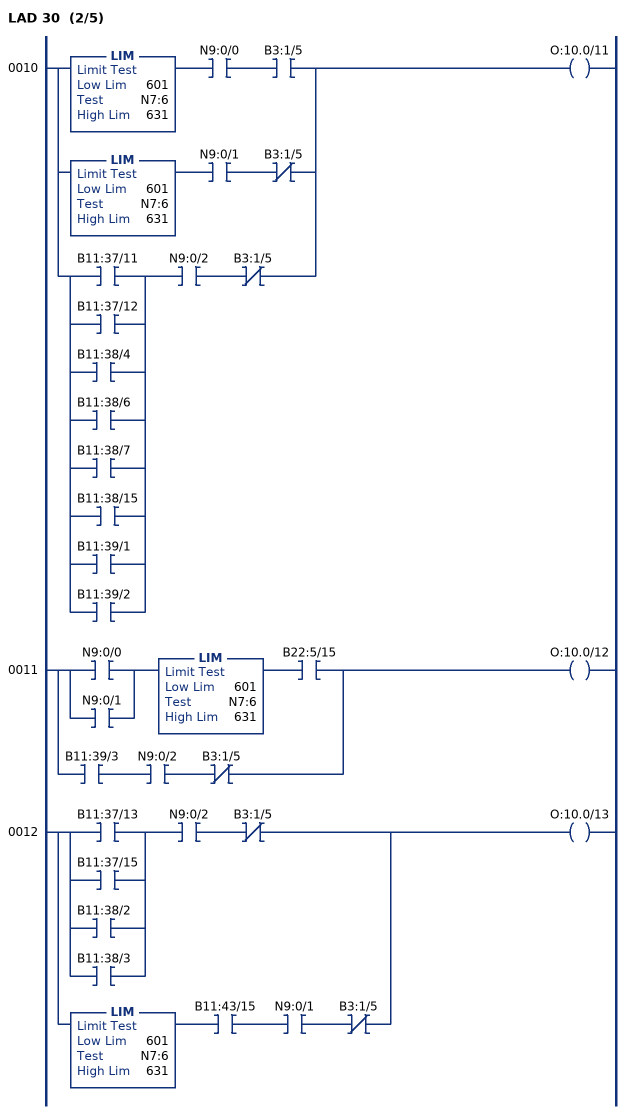
% Rung: 10 %
SOR BST LIM 601 N7:6 631 XIC N9:0/0 XIC B3:1/5 NXB LIM 601 N7:6 631 XIC N9:0/1 XIO B3:1/5 NXB BST XIC B11:37/11 NXB XIC B11:37/12 NXB XIC B11:38/4 NXB XIC B11:38/6 NXB XIC B11:38/7 NXB XIC B11:38/15 NXB XIC B11:39/1 NXB XIC B11:39/2 BND XIC N9:0/2 XIO B3:1/5 BND OTE O:10.0/11 EOR
% Rung: 11 %
SOR BST BST XIC N9:0/0 NXB XIC N9:0/1 BND LIM 601 N7:6 631 XIC B22:5/15 NXB XIC B11:39/3 XIC N9:0/2 XIO B3:1/5 BND OTE O:10.0/12 EOR
% Rung: 12 %
SOR BST BST XIC B11:37/13 NXB XIC B11:37/15 NXB XIC B11:38/2 NXB XIC B11:38/3 BND XIC N9:0/2 XIO B3:1/5 NXB LIM 601 N7:6 631 XIC B11:43/15 XIC N9:0/1 XIO B3:1/5 BND OTE O:10.0/13 EOR

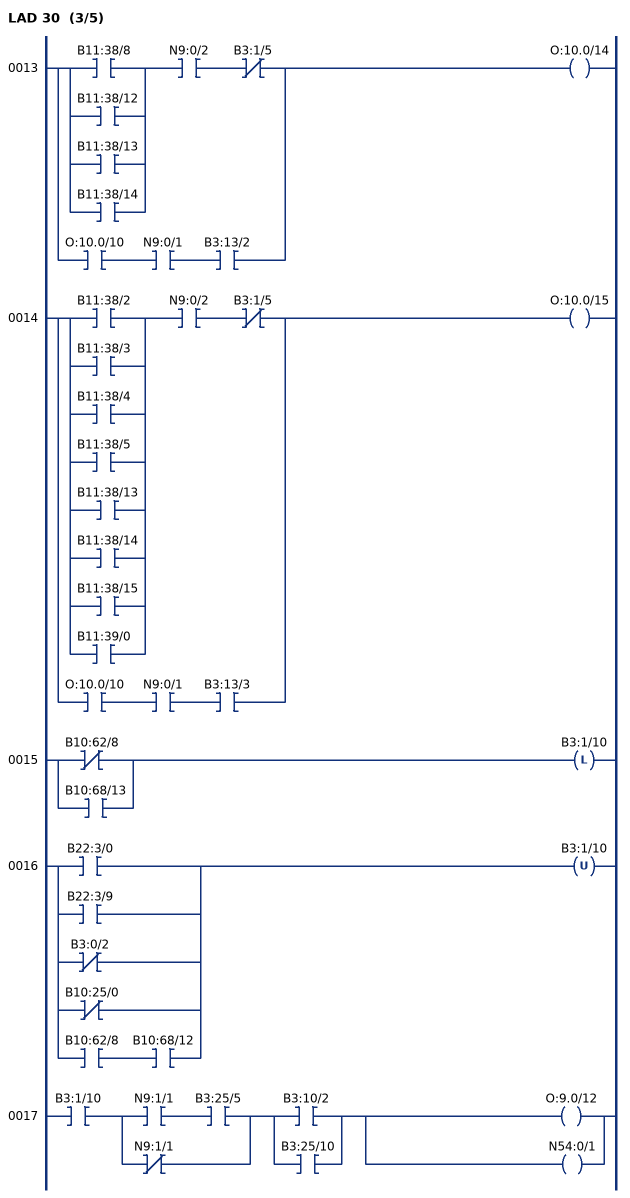
% Rung: 13 %
SOR BST BST XIC B11:38/8 NXB XIC B11:38/12 NXB XIC B11:38/13 NXB XIC B11:38/14 BND XIC N9:0/2 XIO B3:1/5 NXB XIC O:10.0/10 XIC N9:0/1 XIC B3:13/2 BND OTE O:10.0/14 EOR
% Rung: 14 %
SOR BST BST XIC B11:38/2 NXB XIC B11:38/3 NXB XIC B11:38/4 NXB XIC B11:38/5 NXB XIC B11:38/13 NXB XIC B11:38/14 NXB XIC B11:38/15 NXB XIC B11:39/0 BND XIC N9:0/2 XIO B3:1/5 NXB XIC O:10.0/10 XIC N9:0/1 XIC B3:13/3 BND OTE O:10.0/15 EOR
% Rung: 15 %
SOR BST XIO B10:62/8 NXB XIC B10:68/13 BND OTL B3:1/10 EOR
% Rung: 16 %
SOR BST XIC B22:3/0 NXB XIC B22:3/9 NXB XIO B3:0/2 NXB XIO B10:25/0 NXB XIC B10:62/8 XIC B10:68/12 BND OTU B3:1/10 EOR
% Rung: 17 %
SOR XIC B3:1/10 BST XIC N9:1/1 XIC B3:25/5 NXB XIO N9:1/1 BND BST XIC B3:10/2 NXB XIC B3:25/10 BND BST OTE O:9.0/12 NXB OTE N54:0/1 BND EOR

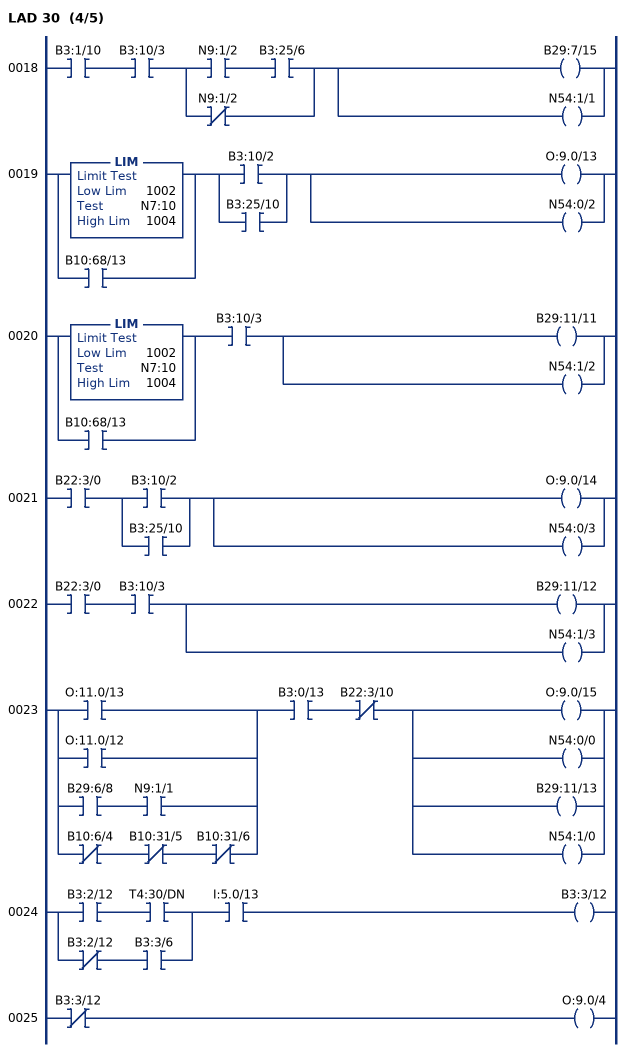
% Rung: 18 %
SOR XIC B3:1/10 XIC B3:10/3 BST XIC N9:1/2 XIC B3:25/6 NXB XIO N9:1/2 BND BST OTE B29:7/15 NXB OTE N54:1/1 BND EOR
% Rung: 19 %
SOR BST LIM 1002 N7:10 1004 NXB XIC B10:68/13 BND BST XIC B3:10/2 NXB XIC B3:25/10 BND BST OTE O:9.0/13 NXB OTE N54:0/2 BND EOR
% Rung: 20 %
SOR BST LIM 1002 N7:10 1004 NXB XIC B10:68/13 BND XIC B3:10/3 BST OTE B29:11/11 NXB OTE N54:1/2 BND EOR
% Rung: 21 %
SOR XIC B22:3/0 BST XIC B3:10/2 NXB XIC B3:25/10 BND BST OTE O:9.0/14 NXB OTE N54:0/3 BND EOR
% Rung: 22 %
SOR XIC B22:3/0 XIC B3:10/3 BST OTE B29:11/12 NXB OTE N54:1/3 BND EOR
% Rung: 23 %
SOR BST BST XIC O:11.0/13 NXB XIC O:11.0/12 BND NXB XIC B29:6/8 XIC N9:1/1 NXB XIO B10:6/4 XIO B10:31/5 XIO B10:31/6 BND XIC B3:0/13 XIO B22:3/10 BST OTE O:9.0/15 NXB OTE N54:0/0 NXB OTE B29:11/13 NXB OTE N54:1/0 BND EOR
% Rung: 24 %
SOR BST XIC B3:2/12 XIC T4:30/DN NXB XIO B3:2/12 XIC B3:3/6 BND XIC I:5.0/13 OTE B3:3/12 EOR
% Rung: 25 %
SOR XIO B3:3/12 OTE O:9.0/4 EOR

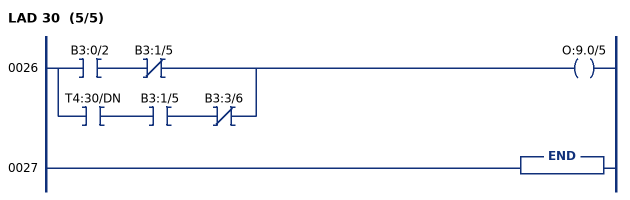
% Rung: 26 %
SOR BST XIC B3:0/2 XIO B3:1/5 NXB XIC T4:30/DN XIC B3:1/5 XIO B3:3/6 BND OTE O:9.0/5 EOR
% Rung: 27 %
SOR END EOR

LADDER 31
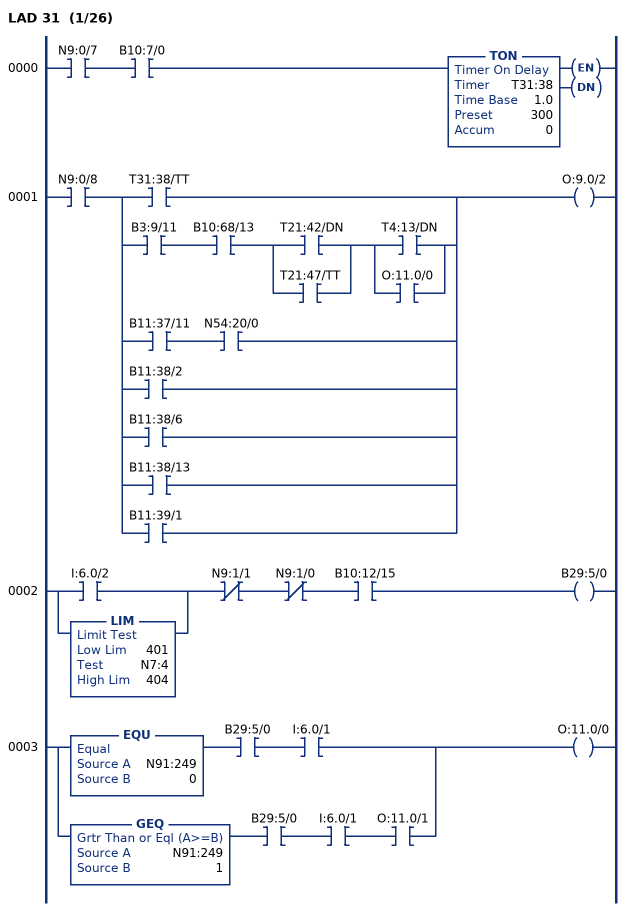
% Rung: 0 %
SOR XIC N9:0/7 XIC B10:7/0 TON T31:38 1.0 300 0 EOR
% Rung: 1 %
SOR XIC N9:0/8 BST XIC T31:38/TT NXB XIC B3:9/11 XIC B10:68/13 BST XIC T21:42/DN NXB XIC T21:47/TT BND BST XIC T4:13/DN NXB XIC O:11.0/0 BND NXB XIC B11:37/11 XIC N54:20/0 NXB XIC B11:38/2 NXB XIC B11:38/6 NXB XIC B11:38/13 NXB XIC B11:39/1 BND OTE O:9.0/2 EOR
% Rung: 2 %
SOR BST XIC I:6.0/2 NXB LIM 401 N7:4 404 BND XIO N9:1/1 XIO N9:1/0 XIC B10:12/15 OTE B29:5/0 EOR
% Rung: 3 %
SOR BST EQU N91:249 0 XIC B29:5/0 XIC I:6.0/1 NXB GEQ N91:249 1 XIC B29:5/0 XIC I:6.0/1 XIC O:11.0/1 BND OTE O:11.0/0 EOR

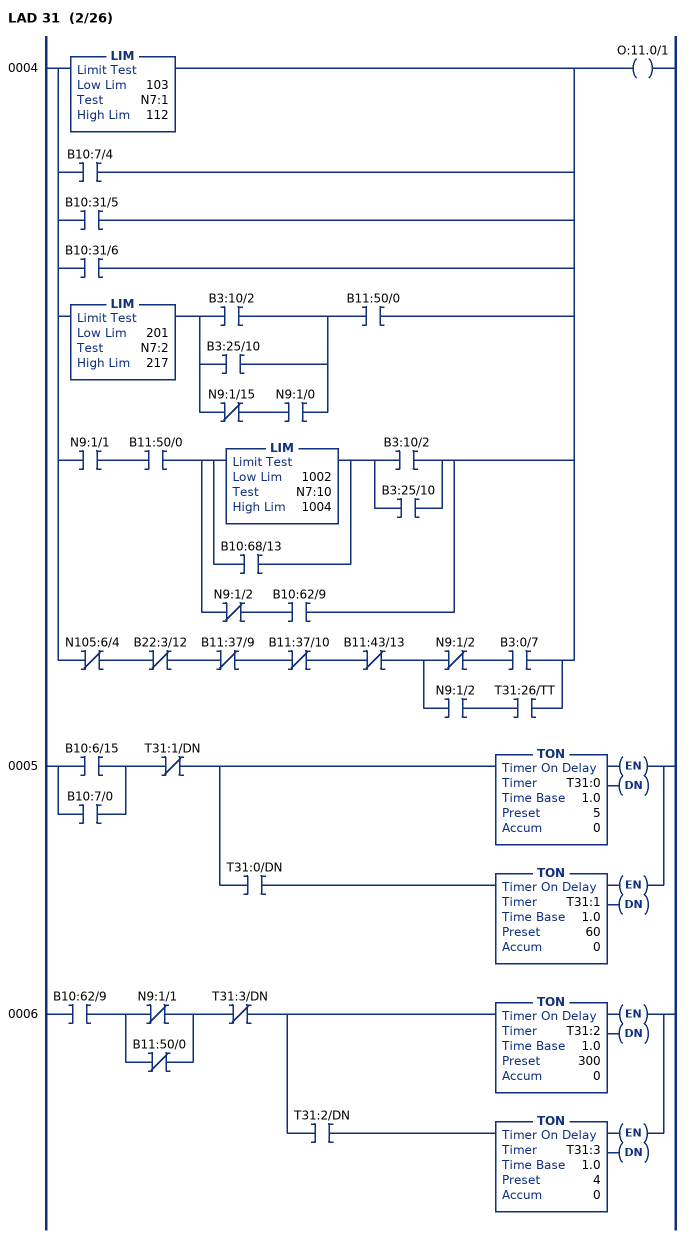
% Rung: 4 %
SOR BST LIM 103 N7:1 112 NXB XIC B10:7/4 NXB XIC B10:31/5 NXB XIC B10:31/6 NXB LIM 201 N7:2 217 BST XIC B3:10/2 NXB XIC B3:25/10 NXB XIO N9:1/15 XIC N9:1/0 BND XIC B11:50/0 NXB XIC N9:1/1 XIC B11:50/0 BST BST LIM 1002 N7:10 1004 NXB XIC B10:68/13 BND BST XIC B3:10/2 NXB XIC B3:25/10 BND NXB XIO N9:1/2 XIC B10:62/9 BND NXB XIO N105:6/4 XIO B22:3/12 XIO B11:37/9 XIO B11:37/10 XIO B11:43/13 BST XIO N9:1/2 XIC B3:0/7 NXB XIC N9:1/2 XIC T31:26/TT BND BND OTE O:11.0/1 EOR
% Rung: 5 %
SOR BST XIC B10:6/15 NXB XIC B10:7/0 BND XIO T31:1/DN BST TON T31:0 1.0 5 0 NXB XIC T31:0/DN TON T31:1 1.0 60 0 BND EOR
% Rung: 6 %
SOR XIC B10:62/9 BST XIO N9:1/1 NXB XIO B11:50/0 BND XIO T31:3/DN BST TON T31:2 1.0 300 0 NXB XIC T31:2/DN TON T31:3 1.0 4 0 BND EOR

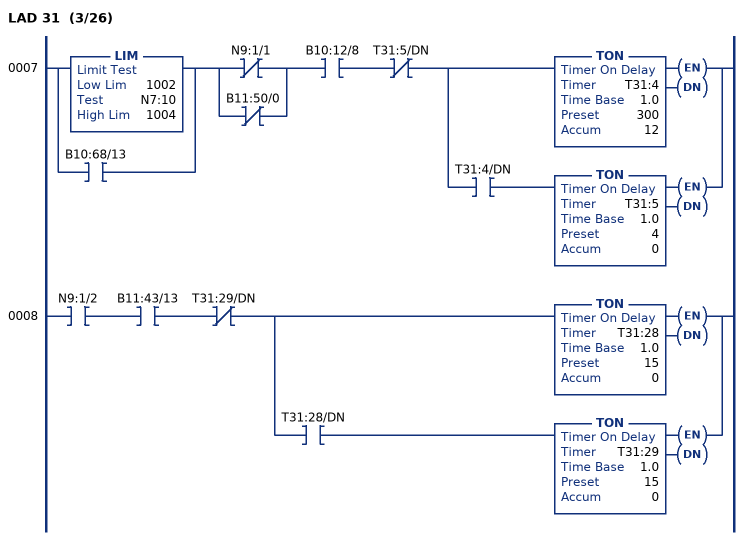
% Rung: 7 %
SOR BST LIM 1002 N7:10 1004 NXB XIC B10:68/13 BND BST XIO N9:1/1 NXB XIO B11:50/0 BND XIC B10:12/8 XIO T31:5/DN BST TON T31:4 1.0 300 12 NXB XIC T31:4/DN TON T31:5 1.0 4 0 BND EOR
% Rung: 8 %
SOR XIC N9:1/2 XIC B11:43/13 XIO T31:29/DN BST TON T31:28 1.0 15 0 NXB XIC T31:28/DN TON T31:29 1.0 15 0 BND EOR

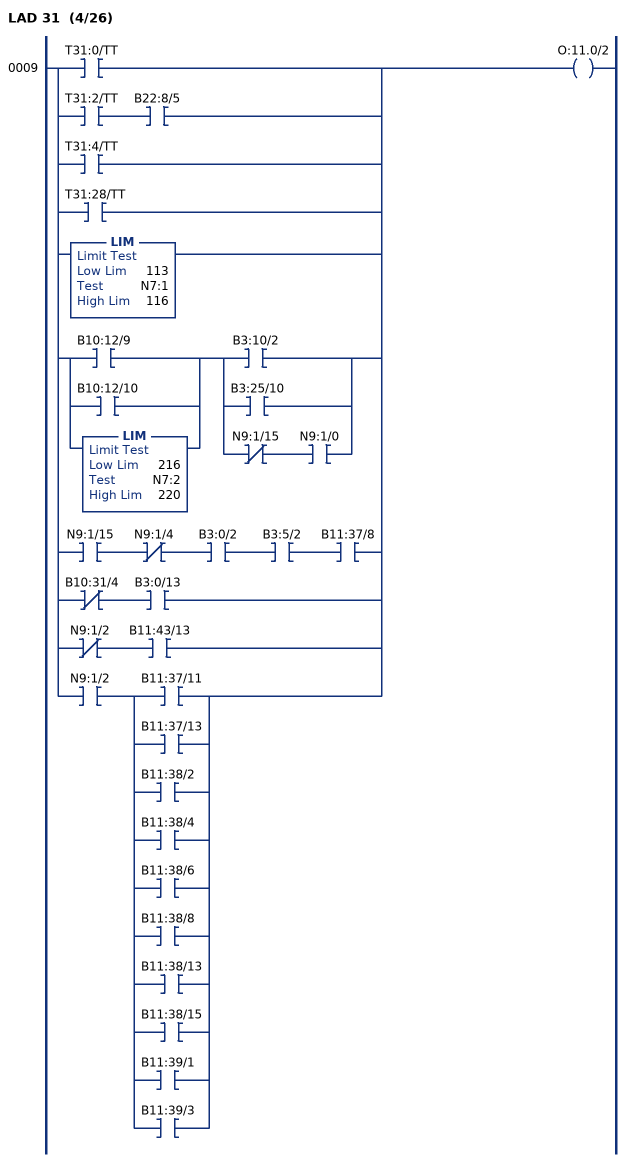
% Rung: 9 %
SOR BST XIC T31:0/TT NXB XIC T31:2/TT XIC B22:8/5 NXB XIC T31:4/TT NXB XIC T31:28/TT NXB LIM 113 N7:1 116 NXB BST XIC B10:12/9 NXB XIC B10:12/10 NXB LIM 216 N7:2 220 BND BST XIC B3:10/2 NXB XIC B3:25/10 NXB XIO N9:1/15 XIC N9:1/0 BND NXB XIC N9:1/15 XIO N9:1/4 XIC B3:0/2 XIC B3:5/2 XIC B11:37/8 NXB XIO B10:31/4 XIC B3:0/13 NXB XIO N9:1/2 XIC B11:43/13 NXB XIC N9:1/2 BST XIC B11:37/11 NXB XIC B11:37/13 NXB XIC B11:38/2 NXB XIC B11:38/4 NXB XIC B11:38/6 NXB XIC B11:38/8 NXB XIC B11:38/13 NXB XIC B11:38/15 NXB XIC B11:39/1 NXB XIC B11:39/3 BND BND OTE O:11.0/2 EOR

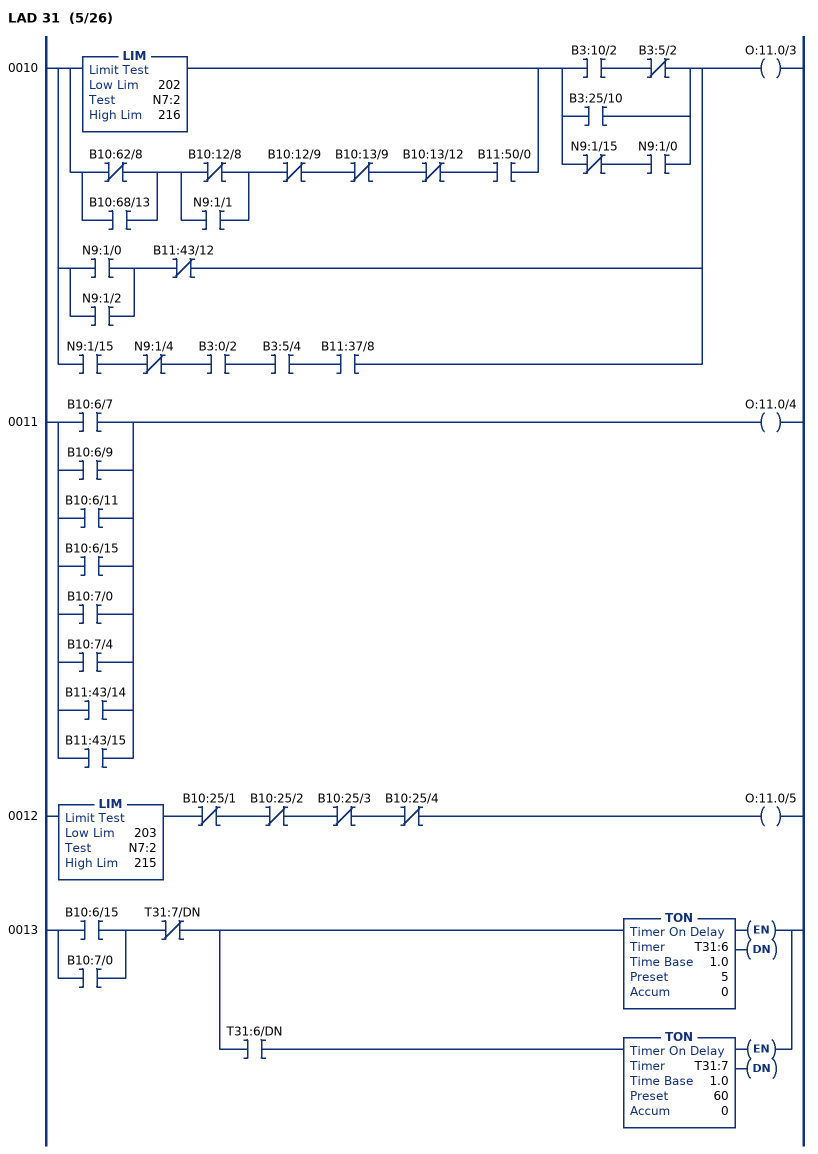
% Rung: 10 %
SOR BST BST LIM 202 N7:2 216 NXB BST XIO B10:62/8 NXB XIC B10:68/13 BND BST XIO B10:12/8 NXB XIC N9:1/1 BND XIO B10:12/9 XIO B10:13/9 XIO B10:13/12 XIC B11:50/0 BND BST XIC B3:10/2 XIO B3:5/2 NXB XIC B3:25/10 NXB XIO N9:1/15 XIC N9:1/0 BND NXB BST XIC N9:1/0 NXB XIC N9:1/2 BND XIO B11:43/12 NXB XIC N9:1/15 XIO N9:1/4 XIC B3:0/2 XIC B3:5/4 XIC B11:37/8 BND OTE O:11.0/3 EOR
% Rung: 11 %
SOR BST XIC B10:6/7 NXB XIC B10:6/9 NXB XIC B10:6/11 NXB XIC B10:6/15 NXB XIC B10:7/0 NXB XIC B10:7/4 NXB XIC B11:43/14 NXB XIC B11:43/15 BND OTE O:11.0/4 EOR
% Rung: 12 %
SOR LIM 203 N7:2 215 XIO B10:25/1 XIO B10:25/2 XIO B10:25/3 XIO B10:25/4 OTE O:11.0/5 EOR
% Rung: 13 %
SOR BST XIC B10:6/15 NXB XIC B10:7/0 BND XIO T31:7/DN BST TON T31:6 1.0 5 0 NXB XIC T31:6/DN TON T31:7 1.0 60 0 BND EOR

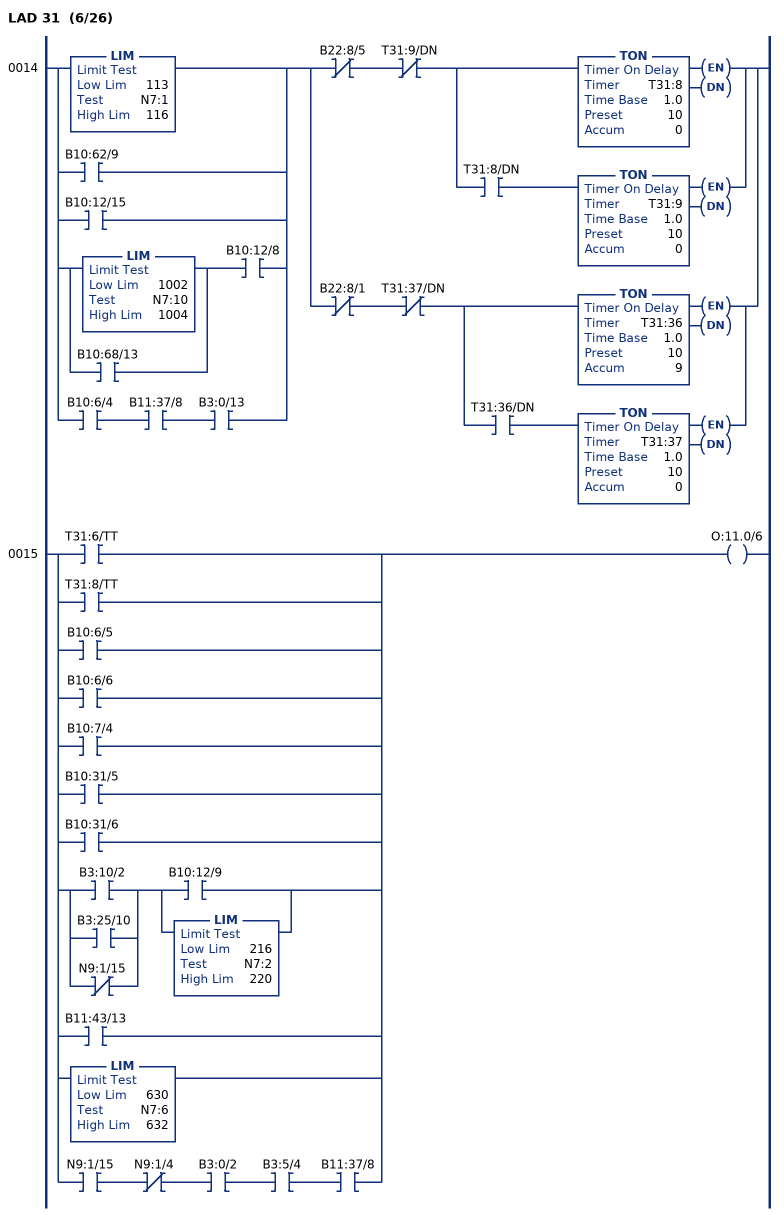
% Rung: 14 %
SOR BST LIM 113 N7:1 116 NXB XIC B10:62/9 NXB XIC B10:12/15 NXB BST LIM 1002 N7:10 1004 NXB XIC B10:68/13 BND XIC B10:12/8 NXB XIC B10:6/4 XIC B11:37/8 XIC B3:0/13 BND BST XIO B22:8/5 XIO T31:9/DN BST TON T31:8 1.0 10 0 NXB XIC T31:8/DN TON T31:9 1.0 10 0 BND NXB XIO B22:8/1 XIO T31:37/DN BST TON T31:36 1.0 10 9 NXB XIC T31:36/DN TON T31:37 1.0 10 0 BND BND EOR
% Rung: 15 %
SOR BST XIC T31:6/TT NXB XIC T31:8/TT NXB XIC B10:6/5 NXB XIC B10:6/6 NXB XIC B10:7/4 NXB XIC B10:31/5 NXB XIC B10:31/6 NXB BST XIC B3:10/2 NXB XIC B3:25/10 NXB XIO N9:1/15 BND BST XIC B10:12/9 NXB LIM 216 N7:2 220 BND NXB XIC B11:43/13 NXB LIM 630 N7:6 632 NXB XIC N9:1/15 XIO N9:1/4 XIC B3:0/2 XIC B3:5/4 XIC B11:37/8 BND OTE O:11.0/6 EOR

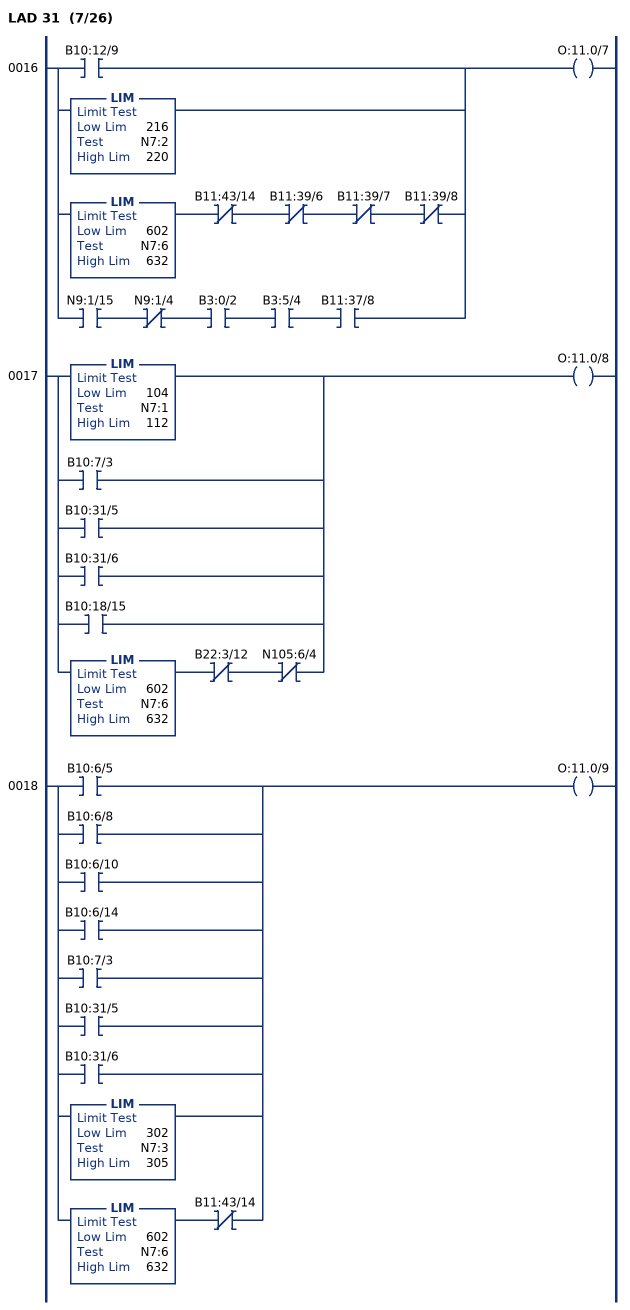
% Rung: 16 %
SOR BST XIC B10:12/9 NXB LIM 216 N7:2 220 NXB LIM 602 N7:6 632 XIO B11:43/14 XIO B11:39/6 XIO B11:39/7 XIO B11:39/8 NXB XIC N9:1/15 XIO N9:1/4 XIC B3:0/2 XIC B3:5/4 XIC B11:37/8 BND OTE O:11.0/7 EOR
% Rung: 17 %
SOR BST LIM 104 N7:1 112 NXB XIC B10:7/3 NXB XIC B10:31/5 NXB XIC B10:31/6 NXB XIC B10:18/15 NXB LIM 602 N7:6 632 XIO B22:3/12 XIO N105:6/4 BND OTE O:11.0/8 EOR
% Rung: 18 %
SOR BST XIC B10:6/5 NXB XIC B10:6/8 NXB XIC B10:6/10 NXB XIC B10:6/14 NXB XIC B10:7/3 NXB XIC B10:31/5 NXB XIC B10:31/6 NXB LIM 302 N7:3 305 NXB LIM 602 N7:6 632 XIO B11:43/14 BND OTE O:11.0/9 EOR

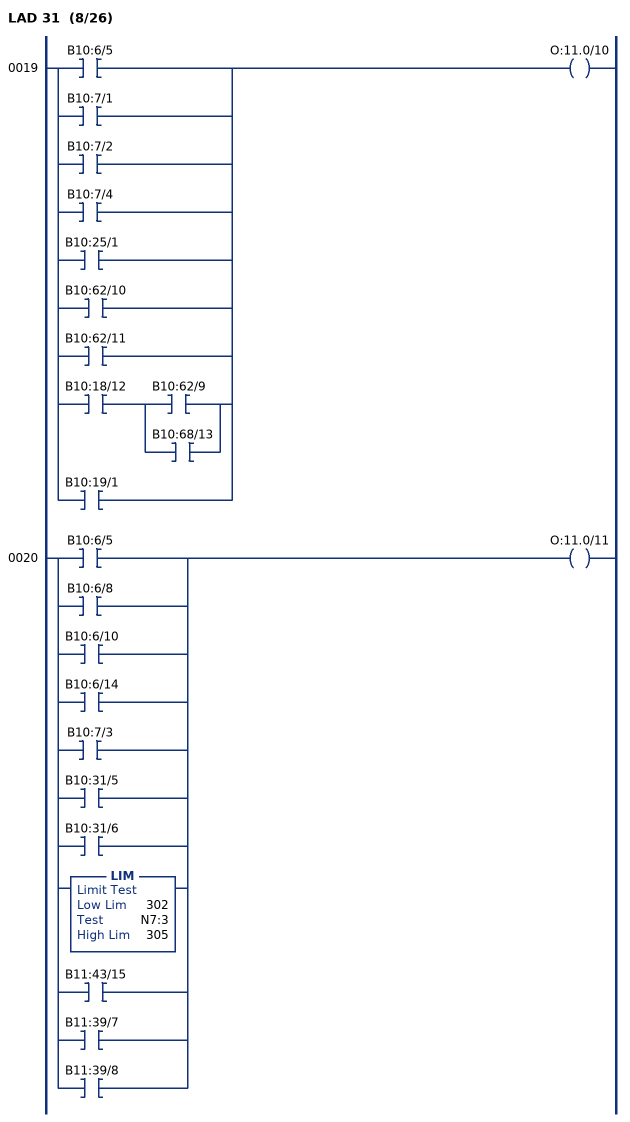
% Rung: 19 %
SOR BST XIC B10:6/5 NXB XIC B10:7/1 NXB XIC B10:7/2 NXB XIC B10:7/4 NXB XIC B10:25/1 NXB XIC B10:62/10 NXB XIC B10:62/11 NXB XIC B10:18/12 BST XIC B10:62/9 NXB XIC B10:68/13 BND NXB XIC B10:19/1 BND OTE O:11.0/10 EOR
% Rung: 20 %
SOR BST XIC B10:6/5 NXB XIC B10:6/8 NXB XIC B10:6/10 NXB XIC B10:6/14 NXB XIC B10:7/3 NXB XIC B10:31/5 NXB XIC B10:31/6 NXB LIM 302 N7:3 305 NXB XIC B11:43/15 NXB XIC B11:39/7 NXB XIC B11:39/8 BND OTE O:11.0/11 EOR

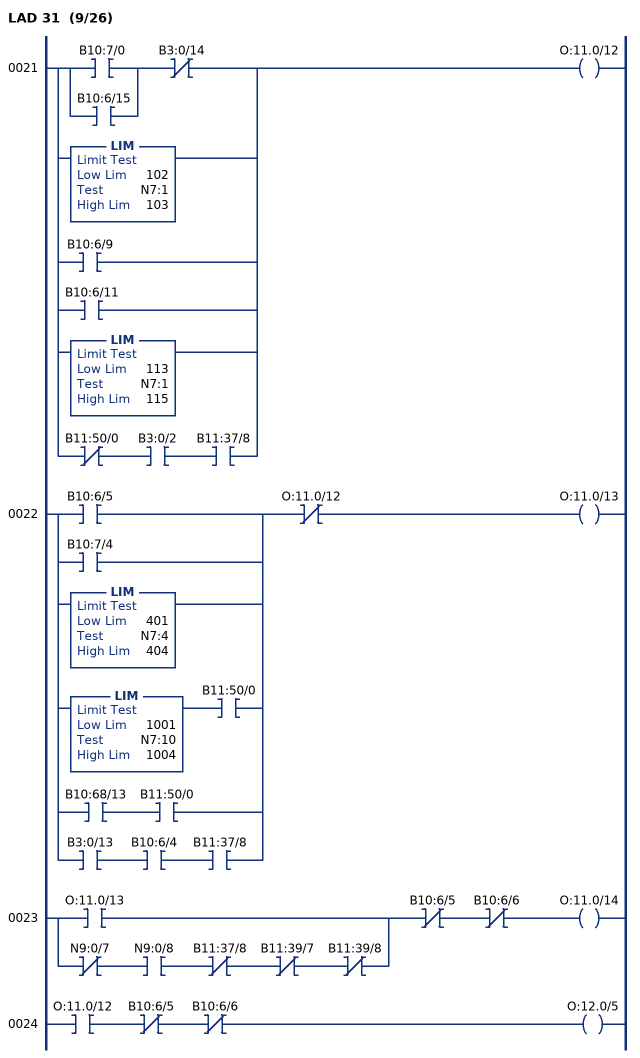
% Rung: 21 %
SOR BST BST XIC B10:7/0 NXB XIC B10:6/15 BND XIO B3:0/14 NXB LIM 102 N7:1 103 NXB XIC B10:6/9 NXB XIC B10:6/11 NXB LIM 113 N7:1 115 NXB XIO B11:50/0 XIC B3:0/2 XIC B11:37/8 BND OTE O:11.0/12 EOR
% Rung: 22 %
SOR BST XIC B10:6/5 NXB XIC B10:7/4 NXB LIM 401 N7:4 404 NXB LIM 1001 N7:10 1004 XIC B11:50/0 NXB XIC B10:68/13 XIC B11:50/0 NXB XIC B3:0/13 XIC B10:6/4 XIC B11:37/8 BND XIO O:11.0/12 OTE O:11.0/13 EOR
% Rung: 23 %
SOR BST XIC O:11.0/13 NXB XIO N9:0/7 XIC N9:0/8 XIO B11:37/8 XIO B11:39/7 XIO B11:39/8 BND XIO B10:6/5 XIO B10:6/6 OTE O:11.0/14 EOR
% Rung: 24 %
SOR XIC O:11.0/12 XIO B10:6/5 XIO B10:6/6 OTE O:12.0/5 EOR

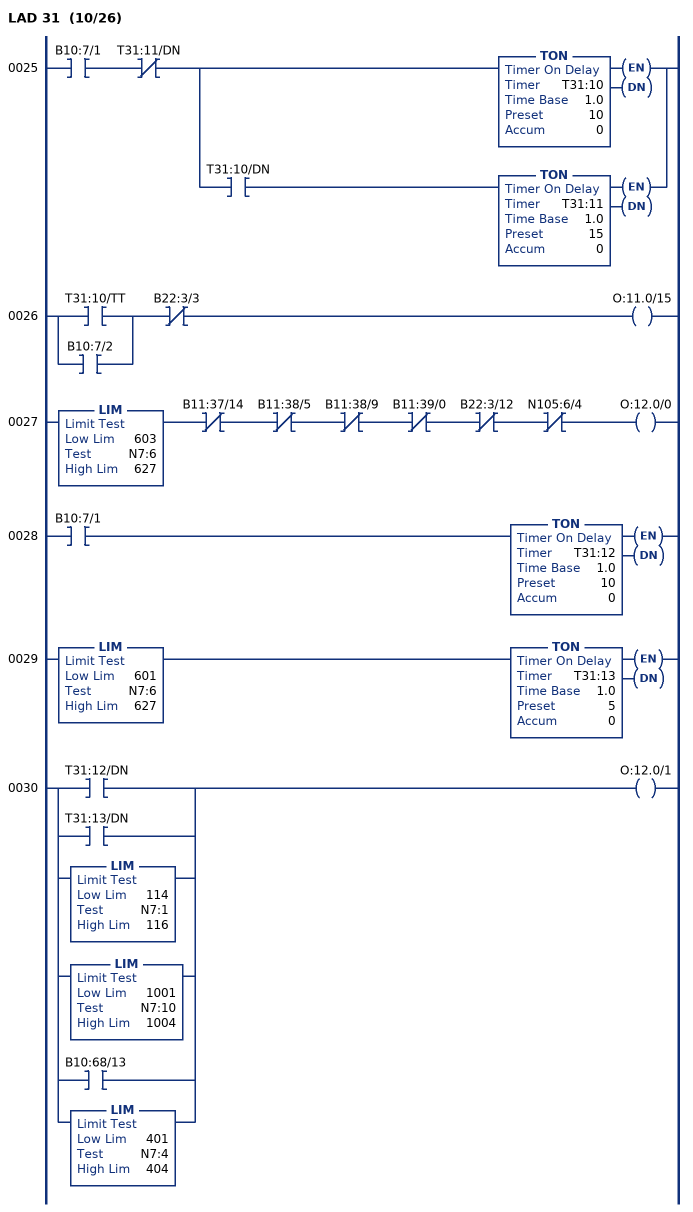
% Rung: 25 %
SOR XIC B10:7/1 XIO T31:11/DN BST TON T31:10 1.0 10 0 NXB XIC T31:10/DN TON T31:11 1.0 15 0 BND EOR
% Rung: 26 %
SOR BST XIC T31:10/TT NXB XIC B10:7/2 BND XIO B22:3/3 OTE O:11.0/15 EOR
% Rung: 27 %
SOR LIM 603 N7:6 627 XIO B11:37/14 XIO B11:38/5 XIO B11:38/9 XIO B11:39/0 XIO B22:3/12 XIO N105:6/4 OTE O:12.0/0 EOR
% Rung: 28 %
SOR XIC B10:7/1 TON T31:12 1.0 10 0 EOR
% Rung: 29 %
SOR LIM 601 N7:6 627 TON T31:13 1.0 5 0 EOR
% Rung: 30 %
SOR BST XIC T31:12/DN NXB XIC T31:13/DN NXB LIM 114 N7:1 116 NXB LIM 1001 N7:10 1004 NXB XIC B10:68/13 NXB LIM 401 N7:4 404 BND OTE O:12.0/1 EOR

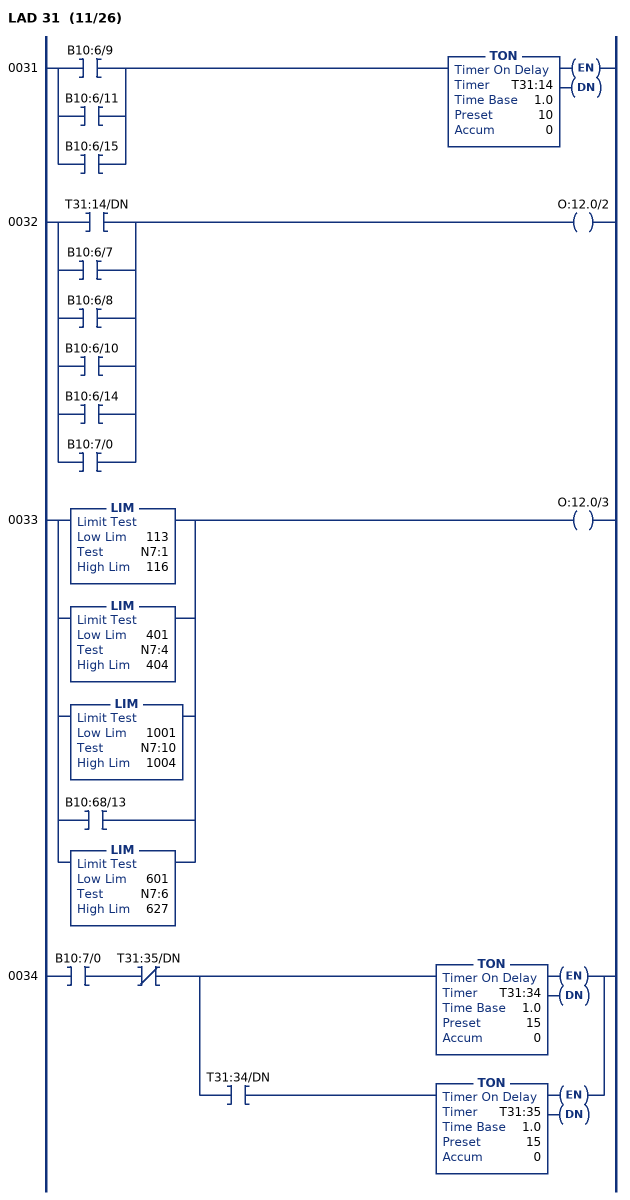
% Rung: 31 %
SOR BST XIC B10:6/9 NXB XIC B10:6/11 NXB XIC B10:6/15 BND TON T31:14 1.0 10 0 EOR
% Rung: 32 %
SOR BST XIC T31:14/DN NXB XIC B10:6/7 NXB XIC B10:6/8 NXB XIC B10:6/10 NXB XIC B10:6/14 NXB XIC B10:7/0 BND OTE O:12.0/2 EOR
% Rung: 33 %
SOR BST LIM 113 N7:1 116 NXB LIM 401 N7:4 404 NXB LIM 1001 N7:10 1004 NXB XIC B10:68/13 NXB LIM 601 N7:6 627 BND OTE O:12.0/3 EOR
% Rung: 34 %
SOR XIC B10:7/0 XIO T31:35/DN BST TON T31:34 1.0 15 0 NXB XIC T31:34/DN TON T31:35 1.0 15 0 BND EOR

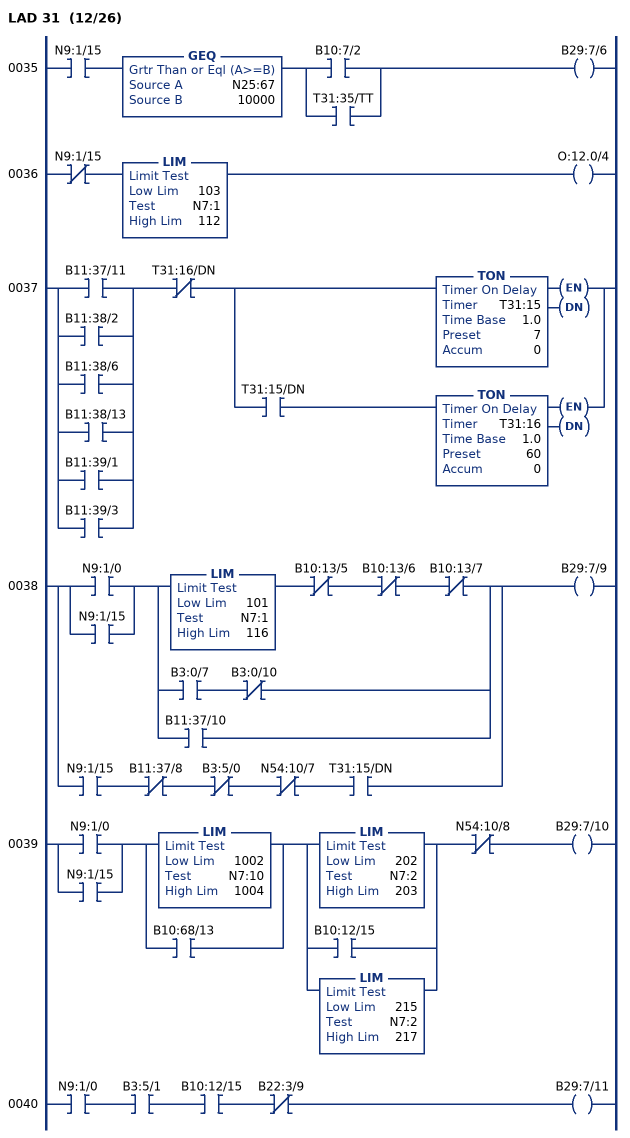
% Rung: 35 %
SOR XIC N9:1/15 GEQ N25:67 10000 BST XIC B10:7/2 NXB XIC T31:35/TT BND OTE B29:7/6 EOR
% Rung: 36 %
SOR XIO N9:1/15 LIM 103 N7:1 112 OTE O:12.0/4 EOR
% Rung: 37 %
SOR BST XIC B11:37/11 NXB XIC B11:38/2 NXB XIC B11:38/6 NXB XIC B11:38/13 NXB XIC B11:39/1 NXB XIC B11:39/3 BND XIO T31:16/DN BST TON T31:15 1.0 7 0 NXB XIC T31:15/DN TON T31:16 1.0 60 0 BND EOR
% Rung: 38 %
SOR BST BST XIC N9:1/0 NXB XIC N9:1/15 BND BST LIM 101 N7:1 116 XIO B10:13/5 XIO B10:13/6 XIO B10:13/7 NXB XIC B3:0/7 XIO B3:0/10 NXB XIC B11:37/10 BND NXB XIC N9:1/15 XIO B11:37/8 XIO B3:5/0 XIO N54:10/7 XIC T31:15/DN BND OTE B29:7/9 EOR
% Rung: 39 %
SOR BST XIC N9:1/0 NXB XIC N9:1/15 BND BST LIM 1002 N7:10 1004 NXB XIC B10:68/13 BND BST LIM 202 N7:2 203 NXB XIC B10:12/15 NXB LIM 215 N7:2 217 BND XIO N54:10/8 OTE B29:7/10 EOR
% Rung: 40 %
SOR XIC N9:1/0 XIC B3:5/1 XIC B10:12/15 XIO B22:3/9 OTE B29:7/11 EOR

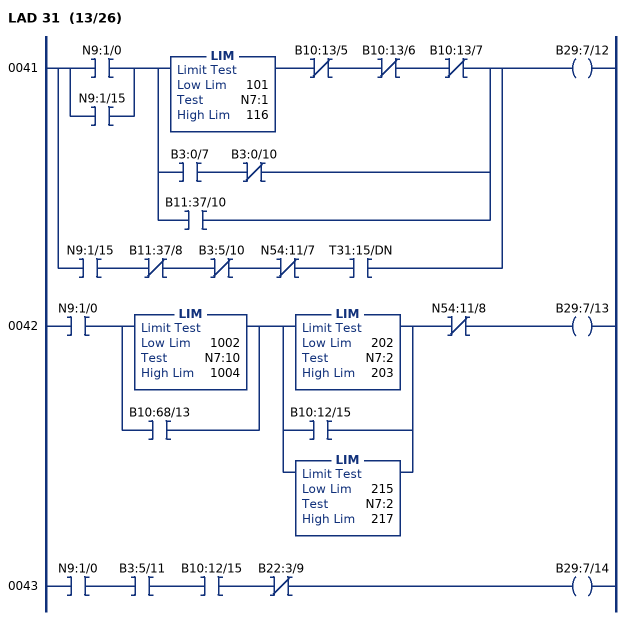
% Rung: 41 %
SOR BST BST XIC N9:1/0 NXB XIC N9:1/15 BND BST LIM 101 N7:1 116 XIO B10:13/5 XIO B10:13/6 XIO B10:13/7 NXB XIC B3:0/7 XIO B3:0/10 NXB XIC B11:37/10 BND NXB XIC N9:1/15 XIO B11:37/8 XIO B3:5/10 XIO N54:11/7 XIC T31:15/DN BND OTE B29:7/12 EOR
% Rung: 42 %
SOR XIC N9:1/0 BST LIM 1002 N7:10 1004 NXB XIC B10:68/13 BND BST LIM 202 N7:2 203 NXB XIC B10:12/15 NXB LIM 215 N7:2 217 BND XIO N54:11/8 OTE B29:7/13 EOR
% Rung: 43 %
SOR XIC N9:1/0 XIC B3:5/11 XIC B10:12/15 XIO B22:3/9 OTE B29:7/14 EOR

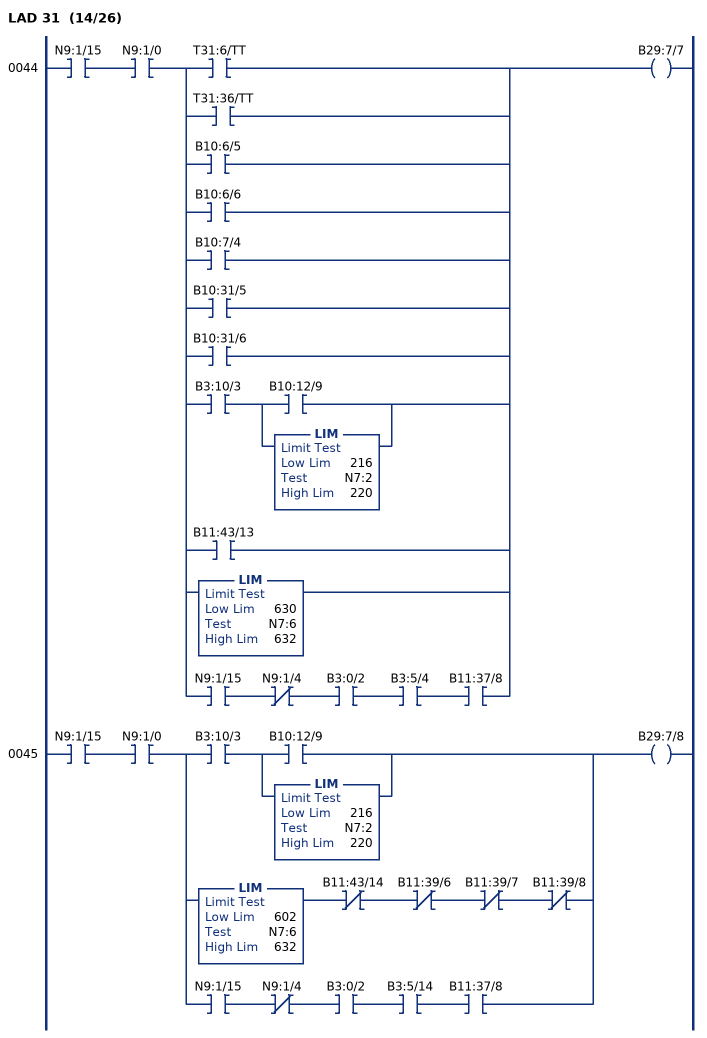
% Rung: 44 %
SOR XIC N9:1/15 XIC N9:1/0 BST XIC T31:6/TT NXB XIC T31:36/TT NXB XIC B10:6/5 NXB XIC B10:6/6 NXB XIC B10:7/4 NXB XIC B10:31/5 NXB XIC B10:31/6 NXB XIC B3:10/3 BST XIC B10:12/9 NXB LIM 216 N7:2 220 BND NXB XIC B11:43/13 NXB LIM 630 N7:6 632 NXB XIC N9:1/15 XIO N9:1/4 XIC B3:0/2 XIC B3:5/4 XIC B11:37/8 BND OTE B29:7/7 EOR
% Rung: 45 %
SOR XIC N9:1/15 XIC N9:1/0 BST XIC B3:10/3 BST XIC B10:12/9 NXB LIM 216 N7:2 220 BND NXB LIM 602 N7:6 632 XIO B11:43/14 XIO B11:39/6 XIO B11:39/7 XIO B11:39/8 NXB XIC N9:1/15 XIO N9:1/4 XIC B3:0/2 XIC B3:5/14 XIC B11:37/8 BND OTE B29:7/8 EOR

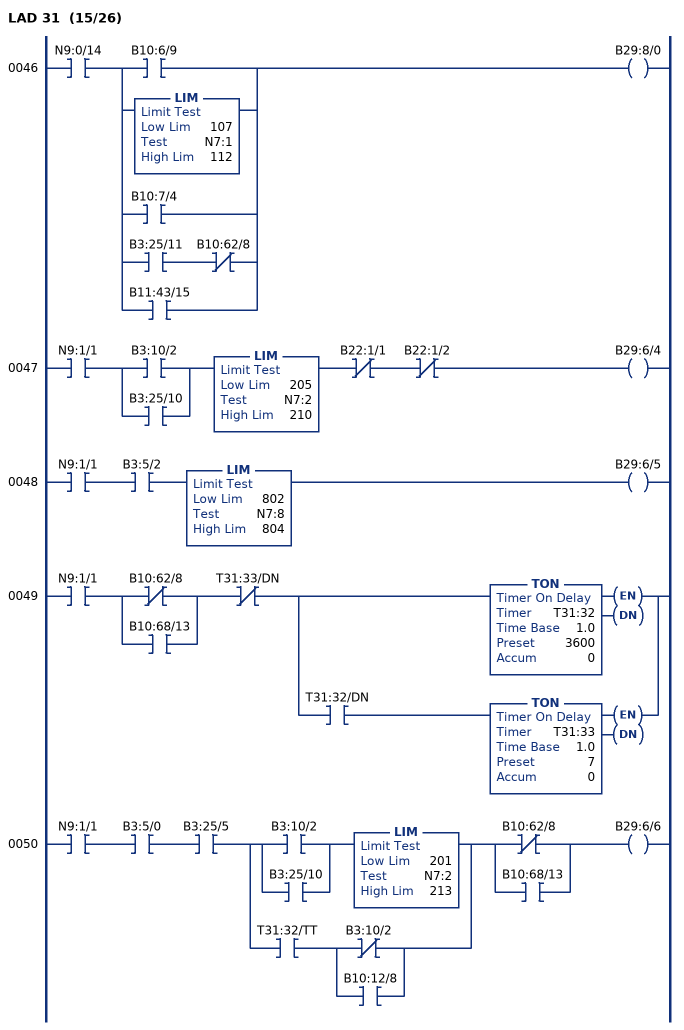
% Rung: 46 %
SOR XIC N9:0/14 BST XIC B10:6/9 NXB LIM 107 N7:1 112 NXB XIC B10:7/4 NXB XIC B3:25/11 XIO B10:62/8 NXB XIC B11:43/15 BND OTE B29:8/0 EOR
% Rung: 47 %
SOR XIC N9:1/1 BST XIC B3:10/2 NXB XIC B3:25/10 BND LIM 205 N7:2 210 XIO B22:1/1 XIO B22:1/2 OTE B29:6/4 EOR
% Rung: 48 %
SOR XIC N9:1/1 XIC B3:5/2 LIM 802 N7:8 804 OTE B29:6/5 EOR
% Rung: 49 %
SOR XIC N9:1/1 BST XIO B10:62/8 NXB XIC B10:68/13 BND XIO T31:33/DN BST TON T31:32 1.0 3600 0 NXB XIC T31:32/DN TON T31:33 1.0 7 0 BND EOR
% Rung: 50 %
SOR XIC N9:1/1 XIC B3:5/0 XIC B3:25/5 BST BST XIC B3:10/2 NXB XIC B3:25/10 BND LIM 201 N7:2 213 NXB XIC T31:32/TT BST XIO B3:10/2 NXB XIC B10:12/8 BND BND BST XIO B10:62/8 NXB XIC B10:68/13 BND OTE B29:6/6 EOR

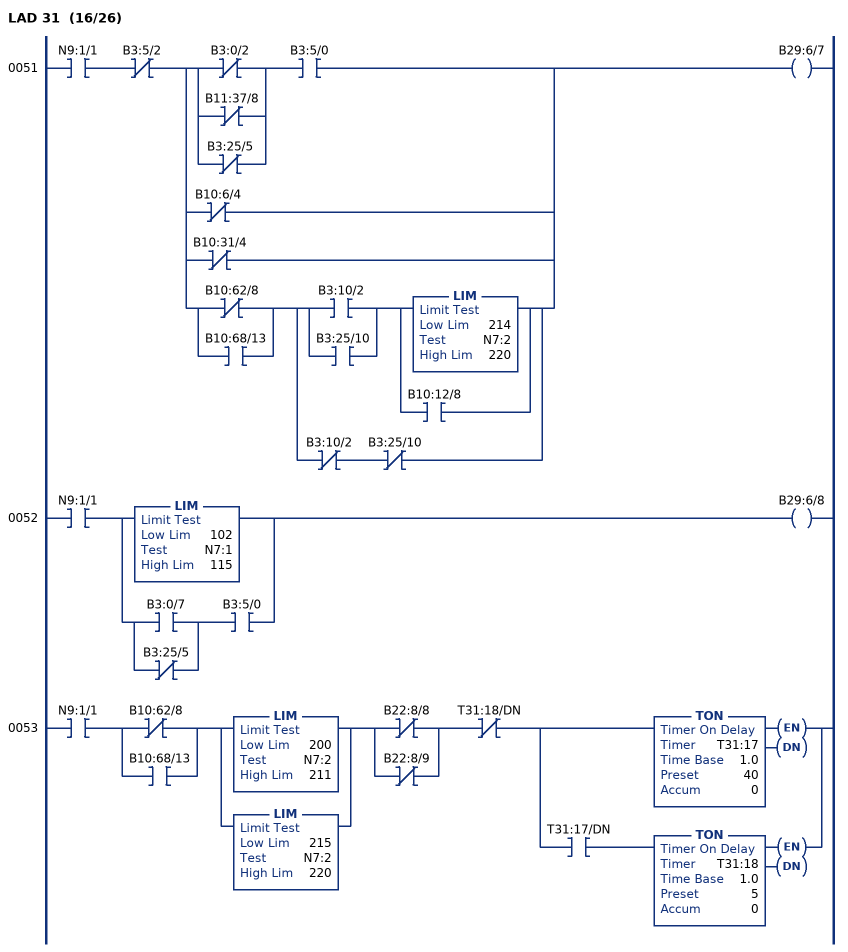
% Rung: 51 %
SOR XIC N9:1/1 XIO B3:5/2 BST BST XIO B3:0/2 NXB XIO B11:37/8 NXB XIO B3:25/5 BND XIC B3:5/0 NXB XIO B10:6/4 NXB XIO B10:31/4 NXB BST XIO B10:62/8 NXB XIC B10:68/13 BND BST BST XIC B3:10/2 NXB XIC B3:25/10 BND BST LIM 214 N7:2 220 NXB XIC B10:12/8 BND NXB XIO B3:10/2 XIO B3:25/10 BND BND OTE B29:6/7 EOR
% Rung: 52 %
SOR XIC N9:1/1 BST LIM 102 N7:1 115 NXB BST XIC B3:0/7 NXB XIO B3:25/5 BND XIC B3:5/0 BND OTE B29:6/8 EOR
% Rung: 53 %
SOR XIC N9:1/1 BST XIO B10:62/8 NXB XIC B10:68/13 BND BST LIM 200 N7:2 211 NXB LIM 215 N7:2 220 BND BST XIO B22:8/8 NXB XIO B22:8/9 BND XIO T31:18/DN BST TON T31:17 1.0 40 0 NXB XIC T31:17/DN TON T31:18 1.0 5 0 BND EOR

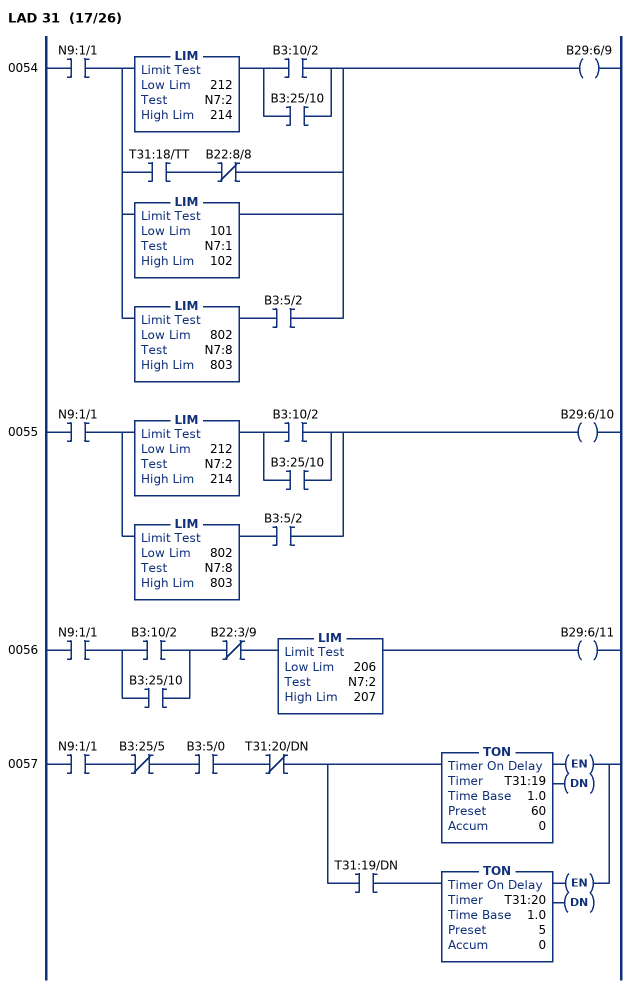
% Rung: 54 %
SOR XIC N9:1/1 BST LIM 212 N7:2 214 BST XIC B3:10/2 NXB XIC B3:25/10 BND NXB XIC T31:18/TT XIO B22:8/8 NXB LIM 101 N7:1 102 NXB LIM 802 N7:8 803 XIC B3:5/2 BND OTE B29:6/9 EOR
% Rung: 55 %
SOR XIC N9:1/1 BST LIM 212 N7:2 214 BST XIC B3:10/2 NXB XIC B3:25/10 BND NXB LIM 802 N7:8 803 XIC B3:5/2 BND OTE B29:6/10 EOR
% Rung: 56 %
SOR XIC N9:1/1 BST XIC B3:10/2 NXB XIC B3:25/10 BND XIO B22:3/9 LIM 206 N7:2 207 OTE B29:6/11 EOR
% Rung: 57 %
SOR XIC N9:1/1 XIO B3:25/5 XIC B3:5/0 XIO T31:20/DN BST TON T31:19 1.0 60 0 NXB XIC T31:19/DN TON T31:20 1.0 5 0 BND EOR

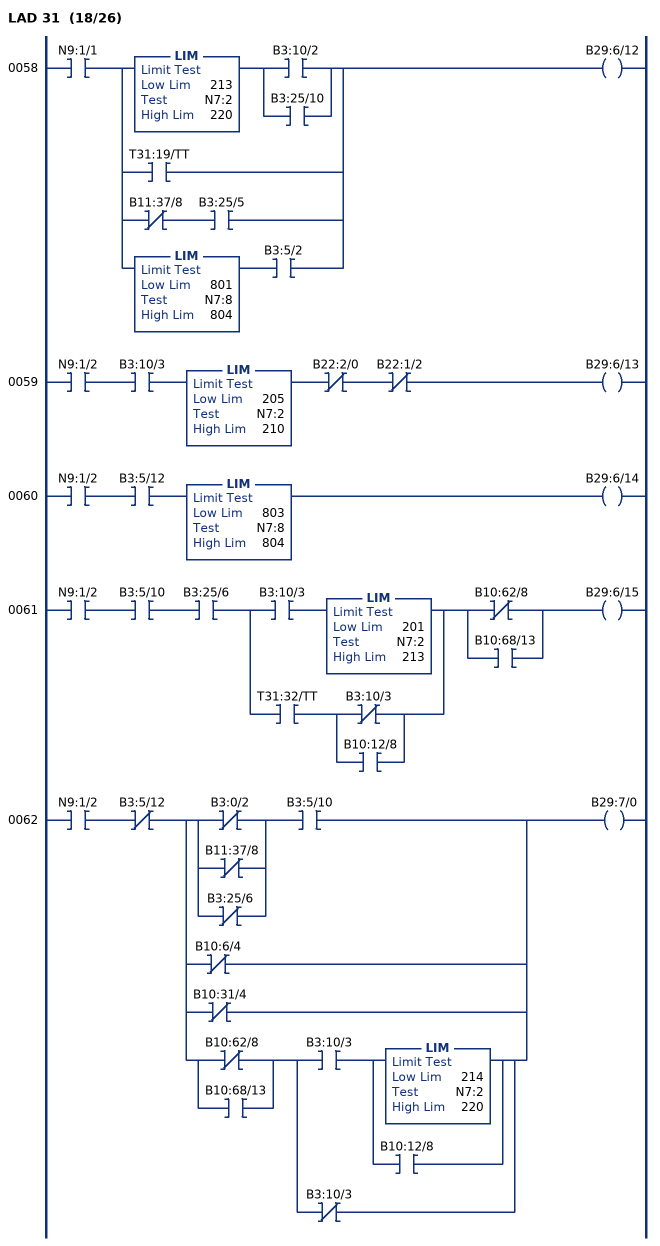
% Rung: 58 %
SOR XIC N9:1/1 BST LIM 213 N7:2 220 BST XIC B3:10/2 NXB XIC B3:25/10 BND NXB XIC T31:19/TT NXB XIO B11:37/8 XIC B3:25/5 NXB LIM 801 N7:8 804 XIC B3:5/2 BND OTE B29:6/12 EOR
% Rung: 59 %
SOR XIC N9:1/2 XIC B3:10/3 LIM 205 N7:2 210 XIO B22:2/0 XIO B22:1/2 OTE B29:6/13 EOR
% Rung: 60 %
SOR XIC N9:1/2 XIC B3:5/12 LIM 803 N7:8 804 OTE B29:6/14 EOR
% Rung: 61 %
SOR XIC N9:1/2 XIC B3:5/10 XIC B3:25/6 BST XIC B3:10/3 LIM 201 N7:2 213 NXB XIC T31:32/TT BST XIO B3:10/3 NXB XIC B10:12/8 BND BND BST XIO B10:62/8 NXB XIC B10:68/13 BND OTE B29:6/15 EOR
% Rung: 62 %
SOR XIC N9:1/2 XIO B3:5/12 BST BST XIO B3:0/2 NXB XIO B11:37/8 NXB XIO B3:25/6 BND XIC B3:5/10 NXB XIO B10:6/4 NXB XIO B10:31/4 NXB BST XIO B10:62/8 NXB XIC B10:68/13 BND BST XIC B3:10/3 BST LIM 214 N7:2 220 NXB XIC B10:12/8 BND NXB XIO B3:10/3 BND BND OTE B29:7/0 EOR

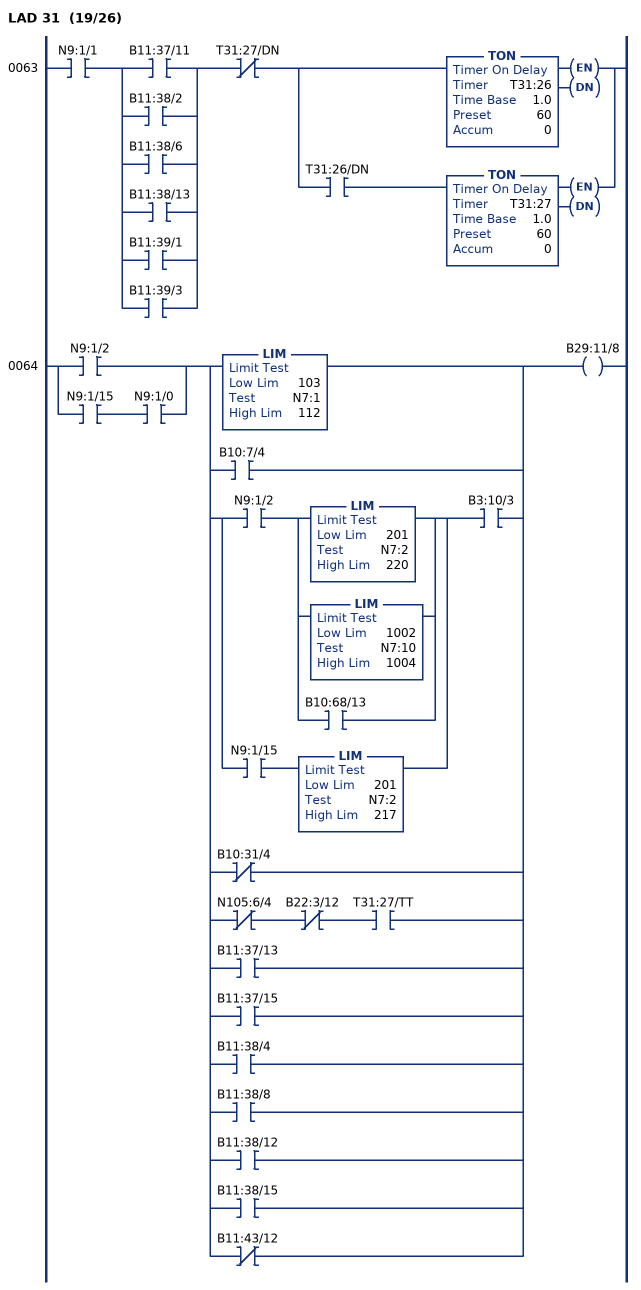
% Rung: 63 %
SOR XIC N9:1/1 BST XIC B11:37/11 NXB XIC B11:38/2 NXB XIC B11:38/6 NXB XIC B11:38/13 NXB XIC B11:39/1 NXB XIC B11:39/3 BND XIO T31:27/DN BST TON T31:26 1.0 60 0 NXB XIC T31:26/DN TON T31:27 1.0 60 0 BND EOR
% Rung: 64 %
SOR BST XIC N9:1/2 NXB XIC N9:1/15 XIC N9:1/0 BND BST LIM 103 N7:1 112 NXB XIC B10:7/4 NXB BST XIC N9:1/2 BST LIM 201 N7:2 220 NXB LIM 1002 N7:10 1004 NXB XIC B10:68/13 BND NXB XIC N9:1/15 LIM 201 N7:2 217 BND XIC B3:10/3 NXB XIO B10:31/4 NXB XIO N105:6/4 XIO B22:3/12 XIC T31:27/TT NXB XIC B11:37/13 NXB XIC B11:37/15 NXB XIC B11:38/4 NXB XIC B11:38/8 NXB XIC B11:38/12 NXB XIC B11:38/15 NXB XIO B11:43/12 BND OTE B29:11/8 EOR

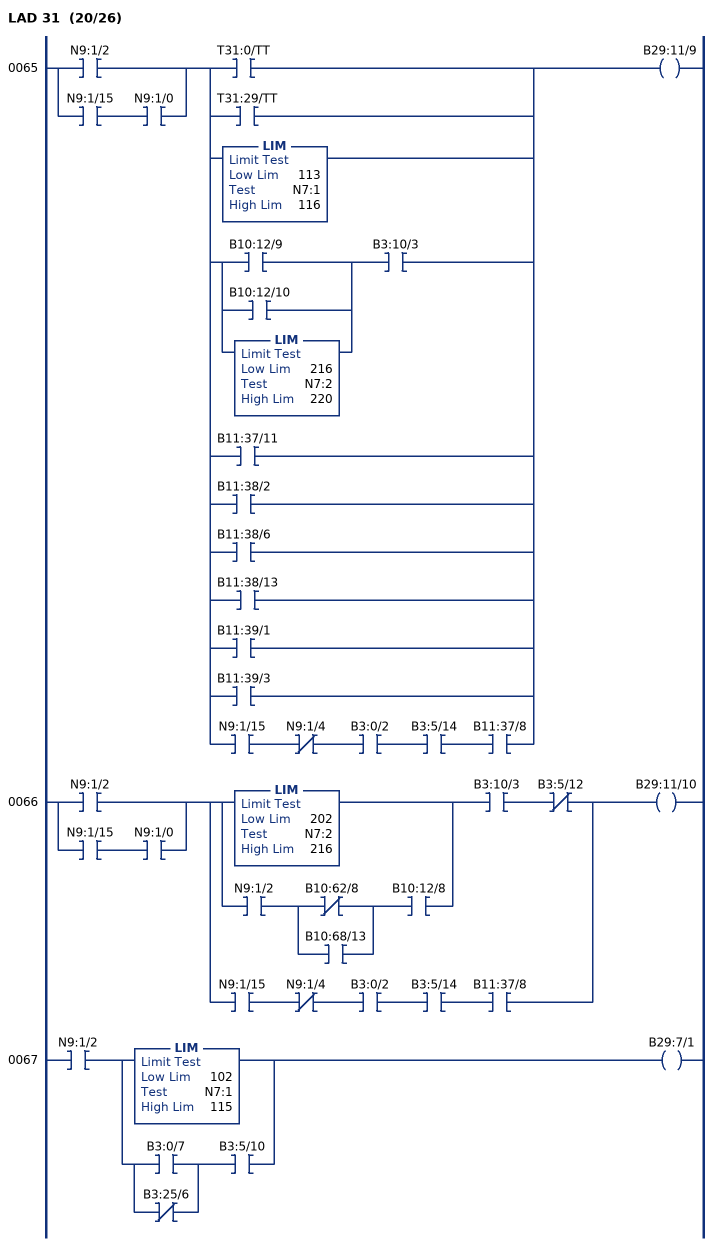
% Rung: 65 %
SOR BST XIC N9:1/2 NXB XIC N9:1/15 XIC N9:1/0 BND BST BST XIC T31:0/TT NXB XIC T31:29/TT NXB LIM 113 N7:1 116 NXB BST XIC B10:12/9 NXB XIC B10:12/10 NXB LIM 216 N7:2 220 BND XIC B3:10/3 NXB XIC B11:37/11 NXB XIC B11:38/2 NXB XIC B11:38/6 NXB XIC B11:38/13 NXB XIC B11:39/1 NXB XIC B11:39/3 BND NXB XIC N9:1/15 XIO N9:1/4 XIC B3:0/2 XIC B3:5/14 XIC B11:37/8 BND OTE B29:11/9 EOR
% Rung: 66 %
SOR BST XIC N9:1/2 NXB XIC N9:1/15 XIC N9:1/0 BND BST BST LIM 202 N7:2 216 NXB XIC N9:1/2 BST XIO B10:62/8 NXB XIC B10:68/13 BND XIC B10:12/8 BND XIC B3:10/3 XIO B3:5/12 NXB XIC N9:1/15 XIO N9:1/4 XIC B3:0/2 XIC B3:5/14 XIC B11:37/8 BND OTE B29:11/10 EOR
% Rung: 67 %
SOR XIC N9:1/2 BST LIM 102 N7:1 115 NXB BST XIC B3:0/7 NXB XIO B3:25/6 BND XIC B3:5/10 BND OTE B29:7/1 EOR

